// Mitsubishi GX Works2 project: 230930-001- exercicios-1   PLC: Q03UDV

PROGRAM MAIN
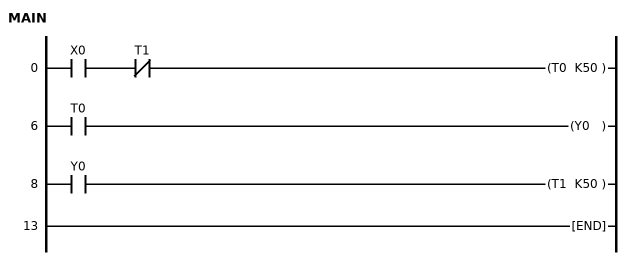
0     LD      X0
      ANI     T1
      OUT     T0 K50
6     LD      T0
      OUT     Y0
8     LD      Y0
      OUT     T1 K50
13    END
END_PROGRAM
